Staubli VAL3: CoreSpeed.pgx

program CoreSpeed(num x_nIndex, mdesc& x_mM)
  local num l_nDist
  local num l_nAngle
begin

  //拐角速度自适应
  //强制把拐角速度给提升
  //只有TxtFile:bBigFileMode 为true时才会调用

   if size(TxtFile:pCut)-1<x_nIndex and TxtFile:nSingleType!=10
    return
  endIf


  l_nDist=distance(TxtFile:pCut[x_nIndex].trsf,TxtFile:pCut[x_nIndex-1].trsf)
  l_nAngle=abs(TxtFile:pCut[x_nIndex].trsf.rx-TxtFile:pCut[x_nIndex-1].trsf.rx)+abs(TxtFile:pCut[x_nIndex].trsf.ry-TxtFile:pCut[x_nIndex-1].trsf.ry)
  l_nAngle=l_nAngle+abs(TxtFile:pCut[x_nIndex].trsf.rz-TxtFile:pCut[x_nIndex-1].trsf.rz)







  //客户可以改距离和相应的拐角大小，加速度大小
  //60指两个点的距离
  //20两个点姿态角度变化大小
  //30强制设置的加速度
  if l_nDist<60 and l_nAngle>20 and x_mM.accel<30
     x_mM.accel=x_mM.decel=30
  endIf



end
